FUNCTION_BLOCK Door (* Composite Function Block Type *)
  (* Standard: 61499-2 *)
  (* Version 0.0, 6/3/2016, Andrei, nxtControl GmbH, template *)
  PACKAGE Main;
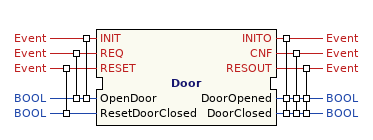
  EVENT_INPUT
    INIT WITH OpenDoor; (* Initialization Request *)
    REQ WITH OpenDoor; (* Normal Execution Request *)
    RESET WITH ResetDoorClosed;
  END_EVENT
  EVENT_OUTPUT
    INITO WITH DoorOpened, DoorClosed; (* Initialization Confirm *)
    CNF WITH DoorOpened, DoorClosed; (* Execution Confirmation *)
    RESOUT WITH DoorOpened, DoorClosed;
  END_EVENT
  VAR_INPUT
    OpenDoor : BOOL; (* Input event qualifier *)
    ResetDoorClosed : BOOL;
  END_VAR
  VAR_OUTPUT
    DoorOpened : BOOL;
    DoorClosed : BOOL;
  END_VAR
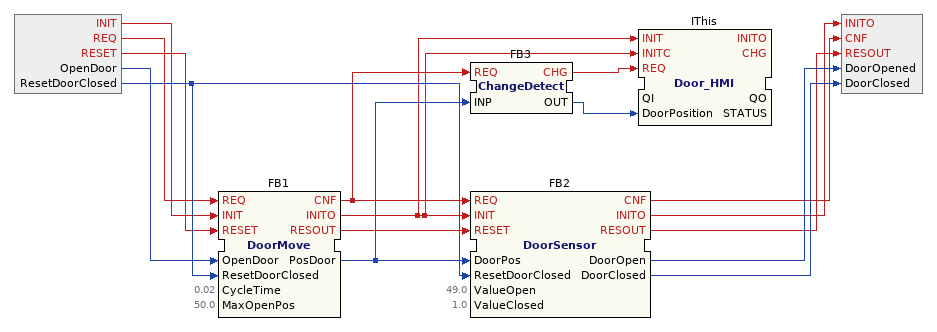
  FBS
    FB3 : ChangeDetect;
    IThis : Door_HMI;
    FB2 : DoorSensor(ValueOpen := 49.0, ValueClosed := 1.0);
    FB1 : DoorMove(CycleTime := 0.02, MaxOpenPos := 50.0);
  END_FBS
  EVENT_CONNECTIONS
    FB1.CNF TO FB2.REQ;
    FB1.INITO TO FB2.INIT;
    FB2.CNF TO CNF;
    FB2.INITO TO INITO;
    REQ TO FB1.REQ;
    INIT TO FB1.INIT;
    FB1.CNF TO FB3.REQ;
    RESET TO FB1.RESET;
    FB1.RESOUT TO FB2.RESET;
    FB1.INITO TO IThis.INIT;
    FB1.INITO TO IThis.INITC;
    FB3.CHG TO IThis.REQ;
    FB2.RESOUT TO RESOUT;
  END_CONNECTIONS
  DATA_CONNECTIONS
    OpenDoor TO FB1.OpenDoor;
    FB1.PosDoor TO FB2.DoorPos;
    FB2.DoorOpen TO DoorOpened;
    FB2.DoorClosed TO DoorClosed;
    FB1.PosDoor TO FB3.INP;
    ResetDoorClosed TO FB2.ResetDoorClosed;
    ResetDoorClosed TO FB1.ResetDoorClosed;
    FB3.OUT TO IThis.DoorPosition;
  END_CONNECTIONS
END_FUNCTION_BLOCK
